// TIA Portal V17 export
// export: Created 2024-08-07T21:43:59.890575Z, ExportSetting WithDefaults, DisplayName Totally Integrated Automation Portal, DisplayVersion V17 Update 7, DisplayName TIA Portal Openness, DisplayVersion V17 Update 7, DisplayName TIA Portal Version Control Interface, DisplayVersion V17, DisplayName SINAMICS Startdrive Advanced, DisplayVersion V17 SP2, DisplayName SINAMICS Startdrive G110M, G120, G120C, G120D, G120P, G115D, DisplayVersion V17 SP2, DisplayName SINAMICS Startdrive G130, G150, S120, S150, SINAMICS MV, S210, DisplayVersion V17 SP2, DisplayName STEP 7 Professional, DisplayVersion V17 Update 7, DisplayName STEP 7 Safety, DisplayVersion V17 Update 6, DisplayName WinCC Advanced / Unified PC, DisplayVersion V17 Update 7
DATA_BLOCK "Manual_DB"   // DB53
VERSION : 0.1
// stored: AutoNumber true, DBAccessibleFromOPCUA true, DBAccessibleFromWebserver true, InstanceOfName Manual, InstanceOfType FB
"Manual"
   // VAR
   //    res : Bool := FALSE;
   //    R_TRIG_MM220bp { S7_SetPoint := 'True'} : R_TRIG;
   //    R_TRIG_MM220wp { S7_SetPoint := 'True'} : R_TRIG;
   //    R_TRIG_MM222bp { S7_SetPoint := 'True'} : R_TRIG;
   //    R_TRIG_MM222wp { S7_SetPoint := 'True'} : R_TRIG;
   //    R_TRIG_MM224bp { S7_SetPoint := 'True'} : R_TRIG;
   //    R_TRIG_MM224wp { S7_SetPoint := 'True'} : R_TRIG;
   // END_VAR
BEGIN
   R_TRIG_MM220bp.CLK := FALSE;
   R_TRIG_MM220bp.Q := FALSE;
   R_TRIG_MM220bp.Stat_Bit := FALSE;
   R_TRIG_MM220wp.CLK := FALSE;
   R_TRIG_MM220wp.Q := FALSE;
   R_TRIG_MM220wp.Stat_Bit := FALSE;
   R_TRIG_MM222bp.CLK := FALSE;
   R_TRIG_MM222bp.Q := FALSE;
   R_TRIG_MM222bp.Stat_Bit := FALSE;
   R_TRIG_MM222wp.CLK := FALSE;
   R_TRIG_MM222wp.Q := FALSE;
   R_TRIG_MM222wp.Stat_Bit := FALSE;
   R_TRIG_MM224bp.CLK := FALSE;
   R_TRIG_MM224bp.Q := FALSE;
   R_TRIG_MM224bp.Stat_Bit := FALSE;
   R_TRIG_MM224wp.CLK := FALSE;
   R_TRIG_MM224wp.Q := FALSE;
   R_TRIG_MM224wp.Stat_Bit := FALSE;
END_DATA_BLOCK
